// TIA Portal V20 export
TYPE "typeEm3MonitoringCmStatus"
// stored: Access Published, Namespace Unit1
   STRUCT
      masterVirtualAxis { ExternalWritable := 'False'} : "LBC_typeAxisControlNodeMonitoring";
      unWinderVirtualAxis { ExternalWritable := 'False'} : "LBC_typeAxisControlNodeMonitoring";
      dancerRegulator { ExternalWritable := 'False'} : "LBC_typeTwoWayActuatorControlNodeMonitoring";
      dancerSafetyPin { ExternalWritable := 'False'} : "LBC_typeDigitalSignalControlNodeMonitoring";
      dancerEncoder { ExternalWritable := 'False'} : "LBC_typeAnalogInputControlNodeMonitoring";
      loadCell { ExternalWritable := 'False'} : "LBC_typeAnalogInputControlNodeMonitoring";
      dancerElectroPneumaticRegulator { ExternalWritable := 'False'} : "LBC_typeAnalogOutputControlNodeMonitoring";
   END_STRUCT;
END_TYPE
